FUNCTION_BLOCK MultiAgentSystemConnector (* JADE WORKER *)
  (* Standard: 61499-1 *)
  (* Version 1.0, 2014-04-22, Ahmed, Fraunhofer IGD *)
  (* Compiler header: package fb.rt; *)
  (* Compiler Java Sun JDK 1.5.0 *)
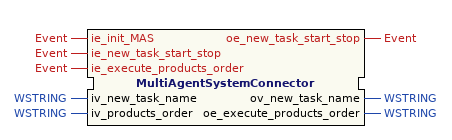
  EVENT_INPUT
    ie_init_MAS;
    ie_new_task_start_stop;
    ie_execute_products_order;
  END_EVENT
  EVENT_OUTPUT
    oe_new_task_start_stop;
  END_EVENT
  VAR_INPUT
    iv_new_task_name : WSTRING;
    iv_products_order : WSTRING;
  END_VAR
  VAR_OUTPUT
    ov_new_task_name : WSTRING;
    oe_execute_products_order : WSTRING;
  END_VAR
END_FUNCTION_BLOCK
